Staubli VAL3: getSizePallet.pgx

public program getSizePallet(string x_sItem, num& x_nSize)
  local string l_sType
  local string l_sKey
  local num i
begin
  //
  // get the size of the collection
  //
  if isDefined(pt:tTraj[x_sItem])
    x_nSize=size(pt:tTraj[x_sItem].tData)
  else
    x_nSize=0
  endIf
end
